// TRUE when nIn > 0; copies nIn to nOut.
FUNCTION IsOk : BOOL
VAR_INPUT
    nIn : Result; // Result to test.
END_VAR
VAR_OUTPUT
    nOut : Result; // Copy of nIn.
END_VAR

IsOk := nIn > 0;
nOut := nIn;

END_FUNCTION

(* stored: Version 1.1.0.1
   POU IsOk: Id {a86826be-b52a-46f1-b35e-fa89d49ee7eb}, SpecialFunc None *)
